ABB RAPID module: Wobj_base_mm_sitevis_cube.mod

MODULE Wobj_base_mm_sitevis_cube
	! Points are read in order of declaration.
  ! Please do not change the order of points!

  LOCAL PERS robtarget pWobj_U_PointX1:=[[1289.542,-192.3507,-459.4274],[0.000332555471686646,-0.289435267448425,0.957173109054565,-0.00684054335579276],[-1,-1,-1,0],[9E+09,9E+09,9E+09,9E+09,9E+09,9E+09]];
	LOCAL PERS robtarget pWobj_U_PointX2:=[[477.4196,-708.0835,-453.8643],[0.000276185455732048,-0.289521455764771,0.957147717475891,-0.00674811797216535],[-1,-1,-1,0],[9E+09,9E+09,9E+09,9E+09,9E+09,9E+09]];
	LOCAL PERS robtarget pWobj_U_PointY1:=[[1633.901,-730.4957,-457.6384],[0.000241211120737717,-0.28953018784523,0.957145214080811,-0.00672532571479678],[-1,-1,-1,0],[9E+09,9E+09,9E+09,9E+09,9E+09,9E+09]];

ENDMODULE
